// TwinCAT 3 PLC project UnitTests
// ProgramVersion: 3.1.4026.21
// libraries:
//   [CoffeeMaker], * (Brandon)
//   Tc2_Standard, * (Beckhoff Automation GmbH)
//   Tc2_System, * (Beckhoff Automation GmbH)
//   TcUnit, * (www.tcunit.org)
// project tree:
//   / PlcTask.TcTTO
//   Test/ FB_HeatingElement_Test.TcPOU, FB_LinkedList_Test.TcPOU, FB_Pump_Test.TcPOU, FB_Scale_Test.TcPOU, FB_TempSensor_Test.TcPOU, PRG_TEST.TcPOU
// (motion and I/O tree: see PLC project plc1)
// real-time tasks:
//   TASK PlcTask: cycle T#10ms, priority 20, ADS port 350
//   TASK PlcTask1: cycle T#10ms, priority 21, ADS port 351

CONFIGURATION UnitTests
    RESOURCE PLC ON TwinCAT3
        TASK PlcTask(INTERVAL := T#10ms, PRIORITY := 21);
        PROGRAM PRG_TEST WITH PlcTask : PRG_TEST;
    END_RESOURCE
END_CONFIGURATION

// ---- Test/PRG_TEST.TcPOU
PROGRAM PRG_TEST
VAR
	fbLinkedList_Test 		: FB_LinkedList_Test;
	fbHeatingElement_Test 	: FB_HeatingElement_Test;
	fbTempSensor_Test		: FB_TempSensor_Test;
	fbScale_Test 			: FB_Scale_Test;
	fbPump_Test				: FB_Pump_Test;
END_VAR

TcUnit.RUN();

END_PROGRAM

// ---- Test/FB_LinkedList_Test.TcPOU
FUNCTION_BLOCK FB_LinkedList_Test EXTENDS FB_TestSuite
VAR
END_VAR

NewListHasLength0();
isEmptyReturnsTrueOnEmptyList();
AddFirstNode();
AddMultipleNodesSameType();
AddMultipleNodesDifferentTypes();
InsertAfterSuccessfully();
RemoveNodeSuccessfully();

METHOD AddFirstNode
VAR
	fbLinkedList : FB_LinkedList;
	
	value : INT := 1;
	getValue : INT;
	
	Actual1 : BOOL;
	Actual2 : UINT;
	Actual3 : INT;
	
	Expected1 : BOOL := FALSE;
	Expected2 : UINT := 1;
	Expected3 : INT := 1;
END_VAR
TEST('AddFirstNode');

fbLinkedList.addValue(value);

Actual1 := fbLinkedList.isEmpty();
AssertEquals(Expected := Expected1, Actual := Actual1, Message := 'isEmpty returns true after adding an item to the list');

Actual2 := fbLinkedList.Length;
AssertEquals(Expected := Expected2, Actual := Actual2, Message := 'Length is not equal to 1 after adding 1 node');

fbLinkedList.getValue(0,getValue);
Actual3 := getValue;
AssertEquals(Expected := Expected3, Actual := Actual3, Message := 'getValue did not return the expected value');

TEST_FINISHED();
END_METHOD

METHOD AddMultipleNodesDifferentTypes
VAR
	fbLinkedList: FB_LinkedList;
	
	intValue 		: INT 		:= 33;
	realValue 		: REAL		:= 3.123;
	stringValue 	: STRING 	:= 'Hello world!';
	
	getInt : INT;
	getReal : REAL;
	getString : STRING;
	
	actualint : INT;
	actualReal : REAL;
	actualString : STRING;
END_VAR
TEST('AddMultipleNodesDifferentTypes');

fbLinkedList.addValue(intValue);
fbLinkedList.addValue(realValue);
fbLinkedList.addValue(stringValue);

fbLinkedList.getValue(0,getInt);
actualInt :=  getInt;
fbLinkedList.getValue(1, getReal);
actualReal := getReal;
fbLinkedList.getValue(2,getString);
actualString := getString;

AssertEquals_INT(expected := intValue, actual := actualInt, message := 'Position 0 was unexpected value');
AssertEquals_REAL(expected := realValue, actual := actualReal, delta := 0.01, message := 'Position 1 was unexpected value');
AssertEquals_STRING(expected := stringValue, actual := actualString, message := 'Position 2 was unexpceted value');

TEST_FINISHED();
END_METHOD

METHOD AddMultipleNodesSameType
VAR
	fbLinkedList : FB_LinkedList;
	intArray : ARRAY [0..4] OF INT := [1,2,3,4,5];
	i : INT;
	Actual: UINT;
	ActualArr: INT;
	Expected: INT := 5;
	ExpectedArr: INT;
END_VAR
TEST('AddMultipleNodesSameType');

FOR i := 0 TO 4 DO
	fbLinkedList.addValue(intArray[i]);
END_FOR

Actual := fbLinkedList.Length;
AssertEquals(Expected := Expected, Actual := Actual, Message := 'Length not equal to 5 after adding 5 nodes');

FOR i := 0 TO 4 DO 
	fbLinkedList.getValue(i, ActualArr);
	ExpectedArr := intArray[i];
	AssertEquals(Expected := ExpectedArr, 
				 Actual := ActualArr, 
				 Message := CONCAT('Index ',CONCAT( INT_TO_STRING(i), CONCAT( ', expected ', CONCAT(INT_TO_STRING(ExpectedArr), CONCAT(', got ', INT_TO_STRING(ActualArr)))))));  
END_FOR

TEST_FINISHED();
END_METHOD

METHOD InsertAfterSuccessfully
VAR
	fbLinkedList : FB_LinkedList;
	initArray : ARRAY [0..4] OF INT := [1,2,3,4,5];
	i : INT;
	
	value : INT := 6;
	
	expectedArray : ARRAY [0..5] OF INT := [1,2,3,4,6,5];
	
	actual : INT;
	expected : INT;
END_VAR
TEST('InsertAfterSuccessfully');

FOR i := 0 TO 4 DO
	fbLinkedList.addValue(initArray[i]);
END_FOR

fbLinkedList.insertAfter(value, 3);

FOR i := 0 TO 4 DO 
	fbLinkedList.getValue(i, actual);
	expected := expectedArray[i];
	AssertEquals(Expected := Expected, Actual := Actual, Message := CONCAT('Index ', CONCAT(INT_TO_STRING(i), ' is not the expcted value'))); 
END_FOR

TEST_FINISHED();
END_METHOD

METHOD isEmptyReturnsTrueOnEmptyList
VAR
	fbLinkedList : FB_LinkedList;
	Expected : BOOL := TRUE;
	Actual: BOOL;
END_VAR
TEST('isEmptyReturnsTrueOnEmptyList');

Actual := fbLinkedList.isEmpty();

AssertEquals(Expected := Expected,
			 Actual := Actual,
			 Message := 'isEmpty() evaluates false on new linked list');
			 
TEST_FINISHED();
END_METHOD

METHOD MoveAfterSuccessfully
VAR
	fbLinkedList : FB_LinkedList;
	initArray : ARRAY [0..4] OF INT := [1,2,3,4,5];
	i : INT;
	
	value : INT := 6;
	
	expectedArray : ARRAY [0..4] OF INT := [1,2,4,3,5];
	
	actual : INT;
	expected : INT;
END_VAR
TEST('MoveAfterSuccessfully');

FOR i := 0 TO 4 DO
	fbLinkedList.addValue(initArray[i]);
END_FOR

fbLinkedList.MoveAfter(2, 3);

FOR i := 0 TO 4 DO 
	fbLinkedList.getValue(i, actual);
	expected := expectedArray[i];
	AssertEquals(Expected := Expected, Actual := Actual, Message := CONCAT('Index ', CONCAT(INT_TO_STRING(i), ' is not the expcted value'))); 
END_FOR

TEST_FINISHED();
END_METHOD

METHOD NewListHasLength0
VAR
	LinkedList : FB_LinkedList;
	Result : UINT;
	ExpectedLength : UINT := 0;
END_VAR
TEST('NewListHasLength0');

Result := LinkedList.Length;

AssertEquals(Expected := ExpectedLength,
			Actual := Result,
			Message := 'New list is not empty');
			
			
	

TEST_FINISHED();
END_METHOD

METHOD OutputReflectsLevel : REFERENCE TO FB_Test
VAR_INPUT
END_VAR
END_METHOD

METHOD RemoveNodeSuccessfully
VAR
	fbLinkedList : FB_LinkedList;
	initArray : ARRAY [0..4] OF INT := [1,2,3,4,5];
	i : INT;
	
	expectedArray : ARRAY [0..3] OF INT := [1,2,4,5];
	
	actual : INT;
	expected : INT;
END_VAR
TEST('RemoveNodeSuccessfully');

FOR i := 0 TO 4 DO
	fbLinkedList.addValue(initArray[i]);
END_FOR

fbLinkedList.remove(2);

FOR i := 0 TO 3 DO 
	fbLinkedList.getValue(i, actual);
	expected := expectedArray[i];
	AssertEquals(Expected := Expected, Actual := Actual, Message := CONCAT('Index ', CONCAT(INT_TO_STRING(i), ' is not the expcted value'))); 
END_FOR

TEST_FINISHED();
END_METHOD

END_FUNCTION_BLOCK

// ---- Test/FB_HeatingElement_Test.TcPOU
FUNCTION_BLOCK FB_HeatingElement_Test EXTENDS FB_TestSuite
VAR
END_VAR

Initialization();
EnableTriggersIdleState();
PowerOffSendsOutput();
PowerOnSendsOutput();
DisableOverridesOutput();

METHOD DisableOverridesOutput : REFERENCE TO FB_Test
VAR_INPUT
END_VAR

VAR
	fbHeatingElement: FB_HeatingElement;
	expectedState: E_State;
	actualState: E_State;
	expectedIsHeating: BOOL;
	actualIsHeating: BOOL;
END_VAR
TEST('DisableOverridesOutput');

fbHeatingElement.Init();
fbHeatingElement.Enable();
fbHeatingElement.PowerOn();
fbHeatingElement.Disable();

expectedState := STOPPED;
actualState := fbHeatingElement.State;
AssertEquals(Expected := expectedState, Actual := actualState, Message := 'State was not STOP following Disable');

expectedIsHeating := FALSE;
actualIsHeating := fbHeatingElement.isHeating;
AssertEquals(Expected := expectedIsHeating, Actual := actualIsHeating, Message := 'isHeating was not FALSE following Disable');

TEST_FINISHED();
END_METHOD

METHOD EnableTriggersIdleState : REFERENCE TO FB_Test
VAR
	fbHeatingElement : FB_HeatingElement;
	expectedState: E_State;
	actualState: E_State;
	actualIsHeating: BOOL;
	expectedIsHeating: BOOL;
END_VAR
TEST('EnableTriggersIdleState');

fbHeatingElement.Init();
fbHeatingElement.Enable();

expectedState := IDLE;
actualState := fbHeatingElement.State;
AssertEquals(Expected := expectedState, Actual := actualState, Message := 'State was not IDLE following enable');

expectedIsHeating := FALSE;
actualIsHeating := fbHeatingElement.isHeating;
AssertEquals(Expected := expectedIsHeating, Actual := actualIsHeating, Message := 'isHeating was not FALSE following enable without powerOn');

TEST_FINISHED();
END_METHOD

METHOD Initialization : REFERENCE TO FB_Test
VAR
	fbHeatingElement : FB_HeatingElement;
	
	expectedState : E_State;
	actualState : E_State;
	
	expectedIsHeating : BOOL := FALSE;
	actualIsHeating : BOOL;
END_VAR
TEST('Initialization');

expectedState := ABORTED;
actualState := fbHeatingElement.State;
AssertEquals(Expected := expectedState, Actual := actualState, Message := 'State was not ABORTED before initialization');

fbHeatingElement.Init();

expectedState := STOPPED;
actualState := fbHeatingElement.State;
AssertEquals(Expected := expectedState, Actual := actualState, Message := 'State was not STOPPED following initialization');

expectedIsHeating := FALSE;
actualIsHeating := fbHeatingElement.isHeating;
AssertEquals(Expected := expectedIsHeating, Actual := actualIsHeating, Message := 'isHeating was not FALSE following initialization');

TEST_FINISHED();
END_METHOD

METHOD PowerOffSendsOutput : REFERENCE TO FB_Test
VAR_INPUT
END_VAR

VAR
	fbHeatingElement: FB_HeatingElement;
	expectedState: E_State;
	actualState: E_State;
	expectedIsHeating: BOOL;
	actualIsHeating: BOOL;
END_VAR
TEST('PowerOffSendsOutput');

fbHeatingElement.Init();
fbHeatingElement.Enable();
fbHeatingElement.PowerOff();

expectedState := IDLE;
actualState := fbHeatingElement.State;
AssertEquals(Expected := expectedState, Actual := actualState, Message := 'State was not IDLE following powerOff');

expectedIsHeating := FALSE;
actualIsHeating := fbHeatingElement.isHeating;
AssertEquals(Expected := expectedIsHeating, Actual := actualIsHeating, Message := 'isHeating was not FALSE following powerOff');

TEST_FINISHED();
END_METHOD

METHOD PowerOnSendsOutput : REFERENCE TO FB_Test
VAR_INPUT
END_VAR

VAR
	fbHeatingElement: FB_HeatingElement;
	expectedState: E_State;
	actualState: E_State;
	expectedIsHeating: BOOL;
	actualIsHeating: BOOL;
END_VAR
TEST('PowerOnSendsOutput');

fbHeatingElement.Init();
fbHeatingElement.Enable();
fbHeatingElement.PowerOn();

expectedState := EXECUTE;
actualState := fbHeatingElement.State;
AssertEquals(Expected := expectedState, Actual := actualState, Message := 'State was not EXECUTE following powerOn');

expectedIsHeating := TRUE;
actualIsHeating := fbHeatingElement.isHeating;
AssertEquals(Expected := expectedIsHeating, Actual := actualIsHeating, Message := 'isHeating was not TRUE following powerOn');

TEST_FINISHED();
END_METHOD

END_FUNCTION_BLOCK

// ---- Test/FB_TempSensor_Test.TcPOU
FUNCTION_BLOCK FB_TempSensor_Test EXTENDS FB_TestSuite
VAR
END_VAR

Initialization();
ValidTemperatureReading();
UpdateRefreshesTemparature();
DetectOutOfRange();
InvalidReadingDoesNotUpdateGoodValue();
SensorRecoversFromFault();

METHOD DetectOutOfRange : REFERENCE TO FB_Test
VAR_INPUT
END_VAR
END_METHOD

METHOD Initialization : REFERENCE TO FB_Test
VAR_INPUT
END_VAR
END_METHOD

METHOD InvalidReadingDoesNotUpdateGoodValue : REFERENCE TO FB_Test
VAR_INPUT
END_VAR
END_METHOD

METHOD SensorRecoversFromFault : REFERENCE TO FB_Test
VAR_INPUT
END_VAR
END_METHOD

METHOD UpdateRefreshesTemparature : REFERENCE TO FB_Test
VAR_INPUT
END_VAR
END_METHOD

METHOD ValidTemperatureReading : REFERENCE TO FB_Test
VAR_INPUT
END_VAR
END_METHOD

END_FUNCTION_BLOCK

// ---- Test/FB_Scale_Test.TcPOU
FUNCTION_BLOCK FB_Scale_Test EXTENDS FB_TestSuite
VAR_INPUT
END_VAR
VAR_OUTPUT
END_VAR
VAR
END_VAR

Initialization();
ValidReading();
UpdateRefreshesWeight();
TareFunction();
WeightReadingAfterTare();
InvalidReadingDetection();
InvalidReadingDoesNotUpdateGoodValue();
ScaleRateCalculation();

METHOD Initialization : REFERENCE TO FB_Test
VAR_INPUT
END_VAR
END_METHOD

METHOD InvalidReadingDetection : REFERENCE TO FB_Test
VAR_INPUT
END_VAR
END_METHOD

METHOD InvalidReadingDoesNotUpdateGoodValue : REFERENCE TO FB_Test
VAR_INPUT
END_VAR
END_METHOD

METHOD ScaleRateCalculation : REFERENCE TO FB_Test
VAR_INPUT
END_VAR
END_METHOD

METHOD TareFunction : REFERENCE TO FB_Test
VAR_INPUT
END_VAR
END_METHOD

METHOD UpdateRefreshesWeight : REFERENCE TO FB_Test
VAR_INPUT
END_VAR
END_METHOD

METHOD ValidReading : REFERENCE TO FB_Test
VAR_INPUT
END_VAR
END_METHOD

METHOD WeightReadingAfterTare : REFERENCE TO FB_Test
VAR_INPUT
END_VAR
END_METHOD

END_FUNCTION_BLOCK

// ---- Test/FB_Pump_Test.TcPOU
FUNCTION_BLOCK FB_Pump_Test EXTENDS FB_TestSuite
VAR_INPUT
END_VAR
VAR_OUTPUT
END_VAR
VAR
END_VAR

Initialize();
EnableTriggersReadyState();
SetFullOutput();
SetZeroOutput();
SetPartialOutput();
DisableOverridesInput();
ClampHighValues();
ClampLowValues();
AutoShutoff();

METHOD AutoShutoff : REFERENCE TO FB_Test
VAR_INPUT
END_VAR
END_METHOD

METHOD ClampHighValues : REFERENCE TO FB_Test
VAR_INPUT
END_VAR
END_METHOD

METHOD ClampLowValues : REFERENCE TO FB_Test
VAR_INPUT
END_VAR
END_METHOD

METHOD DisableOverridesInput : REFERENCE TO FB_Test
VAR_INPUT
END_VAR
END_METHOD

METHOD EnableTriggersReadyState : REFERENCE TO FB_Test
VAR_INPUT
END_VAR
END_METHOD

METHOD Initialize : REFERENCE TO FB_Test
VAR_INPUT
END_VAR
END_METHOD

METHOD SetFullOutput : REFERENCE TO FB_Test
VAR_INPUT
END_VAR
END_METHOD

METHOD SetPartialOutput : REFERENCE TO FB_Test
VAR_INPUT
END_VAR
END_METHOD

METHOD SetZeroOutput : REFERENCE TO FB_Test
VAR_INPUT
END_VAR
END_METHOD

END_FUNCTION_BLOCK
